SUBAPPLICATION SystemTickSender_OPC (* SystemTick-Heartbeat NUR per OPC-UA publizieren, fuer Module ohne eigene VT-Anbindung *)
  (* Standard: 61499-2; Description: Copyright (c) 2026 Meisterschulen am Ostbahnhof This program and the accompanying materials are made available under the terms of the Eclipse Public License 2.0 which is available at https://www.eclipse.org/legal/epl-2.0/ SPDX-License-Identifier: EPL-2.0 *)
  (* Version 1.0, 2026-08-07, Franz Höpfinger, Meisterschulen am Ostbahnhof, initial API and implementation and/or initial documentation *)
  PACKAGE MyLib::sys;
  IMPORT isobus::UT::Q::const::IDs::ID_NULL;
  (* Documentation:
  SystemTick-Heartbeat nur per OPC-UA publizieren
   Schlankste Variante für Module ohne eigene VT-Anbindung: der laufende Tick-Zähler von System_Tick wird direkt per OPC-UA veröffentlicht (ADI_PUBLISH_1, ID_WRITE), ohne lokale VT-Anzeige. Ein anderes Modul mit VT kann diesen Wert per Remote-Subscribe abonnieren und anzeigen, um die Lebendigkeit dieses Moduls zu überwachen.
   Wird zusätzlich eine lokale VT-Anzeige gebraucht, SystemTickSender_ISO_OPC (VT + OPC-UA) bzw. SystemTickSender_ISO (nur VT) verwenden.
  *)
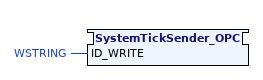
  VAR_INPUT
    ID_WRITE : WSTRING; (* OPC-UA Publish-Key fuer den Tick-Zaehlerstand (fuer Remote-Subscribe durch andere Module) *)
  END_VAR
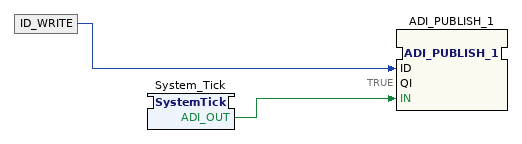
  FBS
    ADI_PUBLISH_1 : adapter::net::ADI_PUBLISH_1(QI := TRUE);
  END_FBS
  SUBAPPS
    System_Tick : MyLib::sys::SystemTick;
  END_SUBAPPS
  DATA_CONNECTIONS
    ID_WRITE TO ADI_PUBLISH_1.ID;
  END_CONNECTIONS
  ADAPTER_CONNECTIONS
    System_Tick.ADI_OUT TO ADI_PUBLISH_1.IN;
  END_CONNECTIONS
END_SUBAPPLICATION
